{attribute 'hide_all_locals' := ''}
{attribute 'FBVisuCreator' := ''}
{attribute 'FBVisuCreatorPrefix' := 'RET_VISU_'}
FUNCTION_BLOCK PT1
VAR_INPUT
	{attribute 'FBVisuCreatorFormatString' := '%1.3f'}
	fX: REAL;
	{attribute 'FBVisuCreatorFormatString' := '%1.3f'}
	fK: REAL;
	{attribute 'FBVisuCreatorFormatString' := '%1.3f'}
	fT: REAL;
	{attribute 'FBVisuCreatorBoolColor' := 'Red'}
	bReset: BOOL;
END_VAR
VAR_OUTPUT
	{attribute 'FBVisuCreatorFormatString' := '%1.3f'}
	fY: REAL;
END_VAR

IF bReset THEN
	reset();
END_IF

IF (fT > 0.0) THEN
	fY := fY + (-fY + fK*fX)/MAX(fT,0.001)*RET_COMMON.fDt;
ELSE
	fY := fX;
END_IF

ACTION reset:
fY := 0.0;
END_ACTION

END_FUNCTION_BLOCK

(* stored: Version 1.1.0.1, ProductVersion 3.1.4024.12
   POU PT1: Id {2f093388-0eb6-4c81-bab3-d16a5cf0b464}, SpecialFunc None
   Action reset: Id {08a2d77e-ca23-4c03-ade9-86ab260f4058} *)
